PROGRAM MAIN
VAR
	fbRead : FB_ModBusReadExample;
	fbWrite : FB_ModBusWriteExample;
	
END_VAR

fbRead();
fbWrite();

END_PROGRAM

(* stored: Version 1.1.0.1, ProductVersion 3.1.4024.16
   POU MAIN: Id {6f8a7c5c-65cf-49f7-b333-8561dc956ed3}, SpecialFunc None *)
